FUNCTION_BLOCK GR_plant_FV (* Basic Function Block Type *)
  (* Standard: 61499-2 *)
  (* Version 0.0, 13/06/2022, Etienne, Schneider Electric, Template *)
  PACKAGE Main;
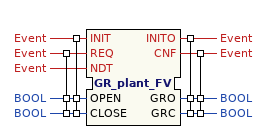
  EVENT_INPUT
    INIT WITH OPEN, CLOSE; (* Initialization Request *)
    REQ WITH OPEN, CLOSE; (* Normal Execution Request *)
    NDT;
  END_EVENT
  EVENT_OUTPUT
    INITO WITH GRO, GRC; (* Initialization Confirm *)
    CNF WITH GRO, GRC; (* Execution Confirmation *)
  END_EVENT
  VAR_INPUT
    OPEN : BOOL;
    CLOSE : BOOL;
  END_VAR
  VAR_OUTPUT
    GRO : BOOL;
    GRC : BOOL;
  END_VAR
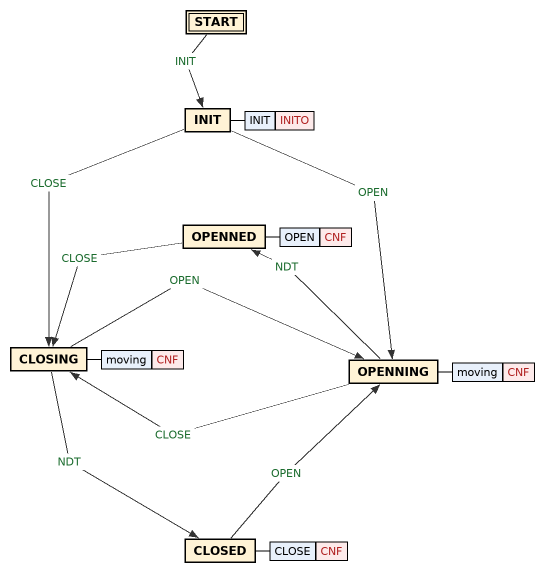
  EC_STATES
    START; (* Initial State *)
    INIT : INIT -> INITO; (* Initialization *)
    OPENNED : OPEN -> CNF;
    CLOSED : CLOSE -> CNF;
    OPENNING : moving -> CNF;
    CLOSING : moving -> CNF;
  END_STATES
  EC_TRANSITIONS
    CLOSING TO CLOSED := NDT;
    CLOSED TO OPENNING := OPEN;
    OPENNING TO OPENNED := NDT;
    OPENNED TO CLOSING := CLOSE;
    START TO INIT := INIT;
    CLOSING TO OPENNING := OPEN;
    OPENNING TO CLOSING := CLOSE;
    INIT TO CLOSING := CLOSE;
    INIT TO OPENNING := OPEN;
  END_TRANSITIONS
  ALGORITHM INIT IN ST: (* Initialization algorithm *)
;
GRO:=FALSE;
GRC:=FALSE;
  END_ALGORITHM
  ALGORITHM OPEN IN ST:
;
GRO := TRUE;
GRC := FALSE;
  END_ALGORITHM
  ALGORITHM moving IN ST:
;
GRO := FALSE;
GRC := FALSE;
  END_ALGORITHM
  ALGORITHM CLOSE IN ST:
;
GRC := TRUE;
GRO := FALSE;
  END_ALGORITHM
  ALGORITHM STOP IN ST:
;
GRO := FALSE;
GRC := FALSE;
  END_ALGORITHM
END_FUNCTION_BLOCK
